PROGRAM POU_readSupvData
VAR
	
	rUpdateRate : TIME := T#900MS;
	sNetId: T_AmsNetId := SUPVams.sNetId;	// '5.30.23.91.1.1';
	nPort: T_AmsPort := SUPVams.nPort; 		// 851

	nFpReadErrorId: UDINT;
	bFpReadError: BOOL;

	
	FB_ReadAmsValue_Fp: FB_ReadAmsValue;
	FB_ReadAmsValue_SPStripperLevel: FB_ReadAmsValue;
	FB_ReadAmsValue_SPPctG: FB_ReadAmsValue;
	
	bLStripReadError: BOOL;
	nFLStripReadErrorId: UDINT;
	bPctGReadError: BOOL;
	nPctGreadErrorId: UDINT;
	FB_ReadAmsValue_SteamValveSP: FB_ReadAmsValue;
	bSteamValveSPReadError: BOOL;
	nSteamValveSPReadErrorId: UDINT;
END_VAR

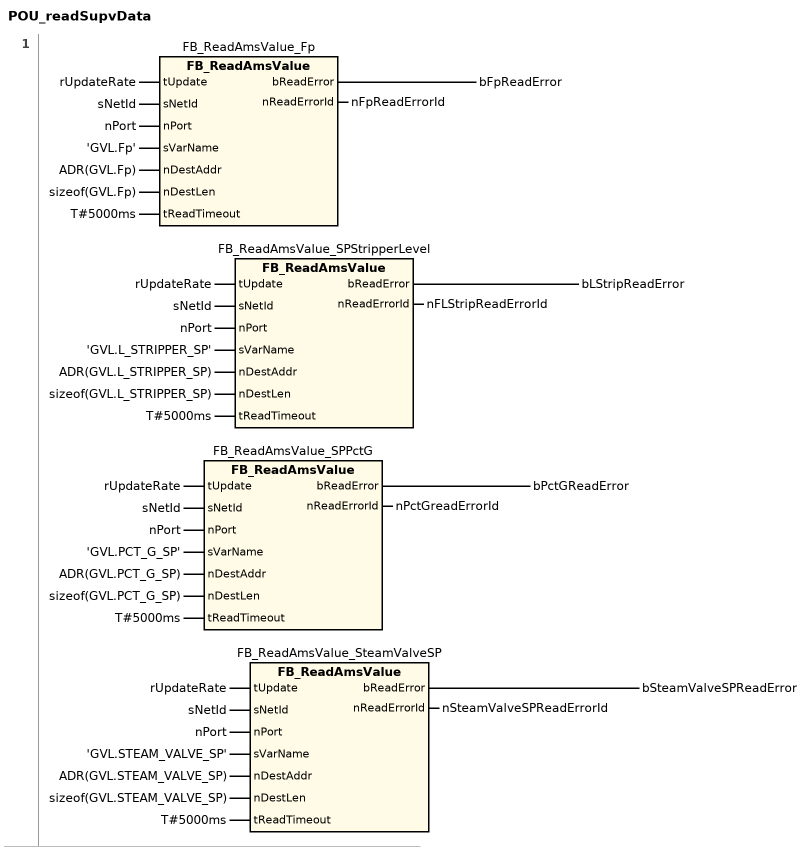
// NETWORK 1
FB_ReadAmsValue_Fp(
    tUpdate := rUpdateRate,
    sNetId := sNetId,
    nPort := nPort,
    sVarName := 'GVL.Fp',
    nDestAddr := ADR(GVL.Fp),
    nDestLen := sizeof(GVL.Fp),
    tReadTimeout := T#5000ms,
    nReadErrorId => nFpReadErrorId); // FB_ReadAmsValue
bFpReadError := FB_ReadAmsValue_Fp.bReadError;
FB_ReadAmsValue_SPStripperLevel(
    tUpdate := rUpdateRate,
    sNetId := sNetId,
    nPort := nPort,
    sVarName := 'GVL.L_STRIPPER_SP',
    nDestAddr := ADR(GVL.L_STRIPPER_SP),
    nDestLen := sizeof(GVL.L_STRIPPER_SP),
    tReadTimeout := T#5000ms,
    nReadErrorId => nFLStripReadErrorId); // FB_ReadAmsValue
bLStripReadError := FB_ReadAmsValue_SPStripperLevel.bReadError;
FB_ReadAmsValue_SPPctG(
    tUpdate := rUpdateRate,
    sNetId := sNetId,
    nPort := nPort,
    sVarName := 'GVL.PCT_G_SP',
    nDestAddr := ADR(GVL.PCT_G_SP),
    nDestLen := sizeof(GVL.PCT_G_SP),
    tReadTimeout := T#5000ms,
    nReadErrorId => nPctGreadErrorId); // FB_ReadAmsValue
bPctGReadError := FB_ReadAmsValue_SPPctG.bReadError;
FB_ReadAmsValue_SteamValveSP(
    tUpdate := rUpdateRate,
    sNetId := sNetId,
    nPort := nPort,
    sVarName := 'GVL.STEAM_VALVE_SP',
    nDestAddr := ADR(GVL.STEAM_VALVE_SP),
    nDestLen := sizeof(GVL.STEAM_VALVE_SP),
    tReadTimeout := T#5000ms,
    nReadErrorId => nSteamValveSPReadErrorId); // FB_ReadAmsValue
bSteamValveSPReadError := FB_ReadAmsValue_SteamValveSP.bReadError;

END_PROGRAM

(* stored: Version 1.1.0.1, ProductVersion 3.1.4024.11
   POU POU_readSupvData: Id {c8dbc9b0-45af-4c0a-8d1c-7f70f78940a5}, SpecialFunc None *)
